TYPE Udt_ParameterId :
STRUCT
	nNumber		: UDINT := 0 	; // parameter number
	sName		: STRING[50] := 'NA' ; // parameter name
	sType		: STRING[4]	:= 'Ppar'	; // parameter type 
	pParameter	: POINTER TO Udt_Parameter ; // pointer to parameter
END_STRUCT
END_TYPE

(* stored: Version 1.1.0.1, ProductVersion 3.1.4024.11
   DUT Udt_ParameterId: Id {781fb137-8d15-4f3c-a209-7913466b6019} *)
